PROGRAM MAIN
VAR
	un : ST_UN;
	
	// Arrays with 'em' universal structure and 'fbEM' containing ST_MACHINE structure which contains of references to fbEM function block
	em : ARRAY[1..Counters.packmlEmLast] OF ST_EM;
	fbEM : ARRAY[1..Counters.packmlEmLast] OF ST_MACHINE;
	
	// Array containing all instances fo fbSliderEM with its own iterator
	SliderEM : ARRAY[1..Counters.SliderEMNo] OF fbSliderEM;
	iSliderEM : DINT := 1;
	
	// Array containing all instances fo fbSliderWithGripperEM with its own iterator
	SliderWithGripperEM : ARRAY[1..Counters.SliderWithGripperEMNo] OF fbSliderWithGripperEM;
	iSliderWithGripperEM : DINT := 1;
	
	// Array containing all instances fo fbXYMoverEM with its own iterator
	XYMoverEM : ARRAY[1..Counters.XYMoverEMNo] OF fbXYMoverEM;
	iXYMoverEM : DINT := 1;
	
	// Flag of initial config, used to set configuration data only once
	InitialConfig : BOOL := TRUE;
	
	// FOR iterator
	i : DINT;
	
	SignalSimSlider: fbSignalSimSlider;
	timer : TON;
END_VAR

IF InitialConfig THEN
	// Specifing module type of each module in array
	em[1].Config.Functionality := E_Function.eSlider;
//	em[2].Config.Functionality := E_Function.eSliderWithGripper;
//	em[3].Config.Functionality := E_Function.eXYMover;

	// FOR loop to specify config for each module
	FOR i := 1 TO Counters.packmlEmLast DO
		em[i].Config.Data.I REF= GVL.aInput[i];
		em[i].Config.Data.Q REF= GVL.aOutput[i];
	
		CASE em[i].Config.Functionality OF
			E_Function.eSlider:
				fbEM[i].fbEM REF= SliderEM[iSliderEM];
				iSliderEM := iSliderEM + 1;
			E_Function.eSliderWithGripper:
				fbEM[i].fbEM REF= SliderWithGripperEM[iSliderWithGripperEM];
				iSliderWithGripperEM := iSliderWithGripperEM + 1;
			E_Function.eXYMover:
				fbEM[i].fbEM REF= XYMoverEM[iXYMoverEM];
				iXYMoverEM := iXYMoverEM + 1;
		END_CASE
	END_FOR
	
	InitialConfig := FALSE;
END_IF

SignalSimSlider(em := em[1], EnableSim := TRUE);

FOR i := 1 TO Counters.packmlEmLast DO
	fbEM[i].fbEM(em := em[i], un := un);
END_FOR

ACTION Init:
// Tutaj planuje przenieść tą inicjalizację a w samym mainie logikę
END_ACTION

END_PROGRAM

(* stored: Version 1.1.0.1, ProductVersion 3.1.4024.12
   POU MAIN: Id {5bccd5a4-76c6-4984-9be1-ff51995fd275}, SpecialFunc None
   Action Init: Id {240e2975-4539-4594-8253-c4c38cfa784d} *)
